Fanuc KAREL source: ka00014.KL

-- PROVISIONAL review KL for V1013-1; original PC SHA256 77dd830446f119687be075e4fe72f16221a65f89c76ed2677c8146b2179c8e38
-- Incomplete behavior may be omitted. Consult companion uncertainty JSON. Do not deploy.
PROGRAM KA00014
%NOLOCKGROUP
VAR
  SRC : REAL
  DST : REAL
BEGIN
  -- UNRESOLVED_PC offsets 5-16; opcodes 2E,23
  -- UNRESOLVED_PC offsets 21-33; opcodes 21,23
  -- UNRESOLVED_PC offsets 38-42; opcodes 7F
END KA00014
